FUNCTION_BLOCK FB_SEL_STRING (* STRING (8-bit) Selection *)
  (* Standard: 61499-1-D.1; Classification: Selection Functions *)
  (* Version 0.1, 2003-11-03, ARM, Tait Control Systems, Completed modification of inputs and output to STRING type *)
  (* Version 0.0, 2002-02-03, JHC, Rockwell Automation, Copied/modified from FB_SEL_WSTRING. *)
  (* Compiler header: package fb.rt.math; *)
  (* Compiler classdef: class FB_SEL_STRING extends FBSelectFunction *)
  (* Compiler Java IBM VisualAge 3.0 *)
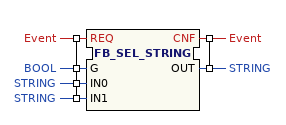
  EVENT_INPUT
    REQ WITH G, IN0, IN1;
  END_EVENT
  EVENT_OUTPUT
    CNF WITH OUT;
  END_EVENT
  VAR_INPUT
    G : BOOL; (* Selector *)
    IN0 : STRING; (* Selected when G=0 *)
    IN1 : STRING; (* Selected when G=1 *)
  END_VAR
  VAR_OUTPUT
    OUT : STRING; (* Selected value *)
  END_VAR
END_FUNCTION_BLOCK
